(* CODESYS project RS485.modbus.20200807.1.project

Project tree, tasks and I/O mapping:
  MIC7001 : Changsha Xiangji-ARM Cortex A9(xilinx zynq7000)-linux, Changsha Xiangji Hiden Technology Co.Ltd, version 3.5.10.40
    application Application
      libraries: CAA Real Time Clock Extern, 3.5.10.0 (CAA Technical Workgroup); CAA Callback Extern, 3.5.11.0 (CAA Technical Workgroup); CAA Can Low Level Imp Extern, 3.5.11.0 (CAA Technical Workgroup); SysMem, 3.5.12.0 (System); CAA DTUtil Extern, 3.5.12.0 (CAA Technical Workgroup); SysTypes2 Interfaces, 3.5.4.0 (System); CAA Types Extern, 3.5.13.0 (CAA Technical Workgroup); Standard, 3.5.14.0 (System); CAA SerialCom, 3.5.15.0 (CAA Technical Workgroup); SysFile, 3.5.15.0 (System); CAA Can Low Level Extern, 3.5.15.0 (CAA Technical Workgroup); CAA Net Base Services, 3.5.15.0 (CAA Technical Workgroup); CAA File, 3.5.15.0 (CAA Technical Workgroup); CAA Memory, 3.5.12.0 (CAA Technical Workgroup)
      task Task (cyclic, interval 200 ms, priority 10) calls COM_modebus_485
      RS485/
        program COM_modebus_485 [ST]
    SoftMotion General Axis Pool
  5ce3da45-db07-42e7-a21c-a00fff4ed8f6|C:\Users\Administrator\Desktop\robotview1.bmp
  5ce3da45-db07-42e7-a21c-a00fff4ed8f6|C:\Users\Administrator\Desktop\robotview2.bmp
  text list GlobalTextList
  5ce3da45-db07-42e7-a21c-a00fff4ed8f6|C:\Users\Administrator\Desktop\1129.bmp
  5ce3da45-db07-42e7-a21c-a00fff4ed8f6|C:\Users\Administrator\Desktop\robotview0.bmp
*)

// MIC7001/Application/RS485/COM_modebus_485
PROGRAM COM_modebus_485
VAR		
	Com1Params: 			ARRAY [1..7] OF COM.PARAMETER;	(* Settings to communicate with the COM Port *)
	hCom: 					CAA.HANDLE;
	ComOpen: 				COM.Open;
	ComClose: 				COM.Close;
	ComWrite: 				COM.Write;
	ComRead: 				COM.Read;	
	
	Snd_Cnt:				CAA.SIZE;

	Rcv_Cnt: 				CAA.SIZE;
	xCom1CloseError: 		BOOL;
	xCom1WriteError: 		BOOL;
	xCom1ReadError: 		BOOL;
	xError:					BOOL;
	
	uiComState: INT := 0;
	ComID:USINT:=8;

	cmdSend:BOOL := FALSE;
	
	Writebuffer:			ARRAY[1..14] OF BYTE;
	Readbuffer: 			ARRAY[1..16] OF BYTE;
    
    crc16 :WORD;
    
    sbwcjy_1:UINT; // 1号传感器的值
    sbwcjy_2:UINT; // 2号传感器的值
END_VAR


//  SW-LDS50A 工业测距传感器, 两个

CASE uiComState OF
	0:
	Com1Params[1].udiParameterId := COM.CAA_Parameter_Constants.udiPort;
	Com1Params[1].udiValue := 8;    //MIC7001的RS485接口为串口8
	Com1Params[2].udiParameterId := COM.CAA_Parameter_Constants.udiBaudrate;
	Com1Params[2].udiValue := 9600;
	Com1Params[3].udiParameterId := COM.CAA_Parameter_Constants.udiParity;
	Com1Params[3].udiValue := INT_TO_UINT(COM.PARITY.NONE);
	Com1Params[4].udiParameterId := COM.CAA_Parameter_Constants.udiStopBits;
	Com1Params[4].udiValue := INT_TO_UINT(COM.STOPBIT.ONESTOPBIT);
	Com1Params[5].udiParameterId := COM.CAA_Parameter_Constants.udiTimeout;
	Com1Params[5].udiValue := 0;
	Com1Params[6].udiParameterId := COM.CAA_Parameter_Constants.udiByteSize;
	Com1Params[6].udiValue := 8;
	Com1Params[7].udiParameterId := COM.CAA_Parameter_Constants.udiBinary;
	Com1Params[7].udiValue := 0;					
	ComOpen(xExecute := TRUE, usiListLength:=UINT_TO_USINT(SIZEOF(Com1Params)/SIZEOF(COM.PARAMETER)),pParameterList:= ADR(Com1Params),hCom=> hCom);			
	IF ComOpen.xError THEN
		uiComState := 32767;
	ELSIF ComOpen.xDone THEN
		uiComState := 10;
	END_IF
	
	10:  // 传感器站号：01  启动一次测量   01 06 00 10 00 01 49 CF  
        Writebuffer[1] := 16#01;
        Writebuffer[2] := 16#06;
        Writebuffer[3] := 16#00;
        Writebuffer[4] := 16#10;
        Writebuffer[5] := 16#00;
        Writebuffer[6] := 16#01;
        
        crc16 := MEM.CRC16_Modbus(ADR(Writebuffer[1]), 6);
        Writebuffer[7] := ANY_TO_BYTE(crc16 MOD 256);
        Writebuffer[8] := ANY_TO_BYTE(crc16/256);
        
		ComWrite(xExecute := TRUE,hCom:= hCom,pBuffer:= ADR(Writebuffer),szSize:= 8);		
		IF ComWrite.xError THEN
			uiComState := 32767;
		END_IF
		IF ComWrite.xDone THEN		
			ComWrite(xExecute := FALSE);
			uiComState := 15;
		END_IF
	
    15:  // 传感器站号：02  启动一次测量   02 06 00 10 00 01   crc_l crc_h
        Writebuffer[1] := 16#02;
        Writebuffer[2] := 16#06;
        Writebuffer[3] := 16#00;
        Writebuffer[4] := 16#10;
        Writebuffer[5] := 16#00;
        Writebuffer[6] := 16#01;
        
        crc16 := MEM.CRC16_Modbus(ADR(Writebuffer[1]), 6);
        Writebuffer[7] := ANY_TO_BYTE(crc16 MOD 256);
        Writebuffer[8] := ANY_TO_BYTE(crc16/256);
        
		ComWrite(xExecute := TRUE,hCom:= hCom,pBuffer:= ADR(Writebuffer),szSize:= 8);		
		IF ComWrite.xError THEN
			uiComState := 32767;
		END_IF
		IF ComWrite.xDone THEN		
			ComWrite(xExecute := FALSE);
			uiComState := 20;
		END_IF   
       
        
	20:  // 发送读取测量值的命令  01 03 00 15 00 02 D5 CF
        Writebuffer[1] := 16#01;
        Writebuffer[2] := 16#03;
        Writebuffer[3] := 16#00;
        Writebuffer[4] := 16#15;
        Writebuffer[5] := 16#00;
        Writebuffer[6] := 16#02;
        
        crc16 := MEM.CRC16_Modbus(ADR(Writebuffer[1]), 6);
        Writebuffer[7] := ANY_TO_BYTE(crc16 MOD 256);
        Writebuffer[8] := ANY_TO_BYTE(crc16/256);
        
		ComWrite(xExecute := TRUE,hCom:= hCom,pBuffer:= ADR(Writebuffer),szSize:= 8);		
		IF ComWrite.xError THEN
			uiComState := 32767;
		END_IF
		IF ComWrite.xDone THEN		
			ComWrite(xExecute := FALSE);
			uiComState := 30;
		END_IF    
    
    30:
        ComRead(xExecute := TRUE,hCom:= hCom, pBuffer:= ADR(Readbuffer), szBuffer:= SIZEOF(Readbuffer));			
        IF ComRead.xError THEN
            uiComState := 32767;
        END_IF
        IF ComRead.xDone THEN
            sbwcjy_1 := ANY_TO_UINT(Readbuffer[6])*256 + ANY_TO_UINT(Readbuffer[7]);
            ComRead(xExecute := FALSE);  // 可以在这里设置断点，观察 Readbuffer 数组中的值
            uiComState := 40;   // 读取成功， 处理下一个传感器
        END_IF
	
     40:  // 发送读取测量值的命令  02 03 00 15 00 02 crc_l crc_h
        Writebuffer[1] := 16#02;
        Writebuffer[2] := 16#03;
        Writebuffer[3] := 16#00;
        Writebuffer[4] := 16#15;
        Writebuffer[5] := 16#00;
        Writebuffer[6] := 16#02;
        
        crc16 := MEM.CRC16_Modbus(ADR(Writebuffer[1]), 6);
        Writebuffer[7] := ANY_TO_BYTE(crc16 MOD 256);
        Writebuffer[8] := ANY_TO_BYTE(crc16/256);
        
		ComWrite(xExecute := TRUE,hCom:= hCom,pBuffer:= ADR(Writebuffer),szSize:= 8);		
		IF ComWrite.xError THEN
			uiComState := 32767;
		END_IF
		IF ComWrite.xDone THEN		
			ComWrite(xExecute := FALSE);
			uiComState := 50;
		END_IF	

    50:
        ComRead(xExecute := TRUE,hCom:= hCom, pBuffer:= ADR(Readbuffer), szBuffer:= SIZEOF(Readbuffer));			
        IF ComRead.xError THEN
            uiComState := 32767;
        END_IF
        IF ComRead.xDone THEN
            sbwcjy_2 := ANY_TO_UINT(Readbuffer[6])*256 + ANY_TO_UINT(Readbuffer[7]);
            ComRead(xExecute := FALSE);  // 可以在这里设置断点，观察 Readbuffer 数组中的值
            uiComState := 20;   // 读取成功， 处理下一个传感器
        END_IF        
        
        
	32767:	
    
END_CASE

END_PROGRAM
